// TIA Portal V20 export
DATA_BLOCK "ControlNodes"   // DB115
// stored: MemoryReserve 100, Namespace Unit1.Em7
   VAR
      em { ExternalWritable := 'False'} : "LAF_typeEmControlNode";
      cm { ExternalWritable := 'False'} : "Unit1.Em7.typeCmControlNode";
      citiMap : "LER_OEM_Data";
      conveyor { ExternalWritable := 'False'} : "Unit1.Em7.typeSequenceControlNodeConveyor";
      ngKicker { ExternalWritable := 'False'} : "Unit1.Em7.typeSequenceControlNodeNgKicker";
      passKicker { ExternalWritable := 'False'} : "Unit1.Em7.typeSequenceControlNodePassKicker";
      qrReaderSTK1 { ExternalWritable := 'False'} : "Unit1.Em7.typeSequenceControlNodeQrReadSTK1";
      qrReaderSTK2 { ExternalWritable := 'False'} : "Unit1.Em7.typeSequenceControlNodeQrReadSTK2";
      InterfaceSTK1 { ExternalWritable := 'False'} : "Unit1.Em7.typeSequenceControlNodeInterafceSTK1";
      InterfaceSTK2 { ExternalWritable := 'False'} : "Unit1.Em7.typeSequenceControlNodeInterafceSTK2";
   END_VAR
   VAR RETAIN
      cmNgKickerAxisZ { ExternalWritable := 'False'} : "LBC_typeAxisControlNode";
      cmPassKickerAxisZ { ExternalWritable := 'False'} : "LBC_typeAxisControlNode";
      cmCutConveyorAxisB { ExternalWritable := 'False'} : "LBC_typeAxisControlNode";
      cmNgConveyorAxisB { ExternalWritable := 'False'} : "LBC_typeAxisControlNode";
      cmStack1ConveyorAxisB { ExternalWritable := 'False'} : "LBC_typeAxisControlNode";
      cmStack2ConveyorAxisB { ExternalWritable := 'False'} : "LBC_typeAxisControlNode";
      cmConveyorVirtualAxisB { ExternalWritable := 'False'} : "LBC_typeAxisControlNode";
      cmCutConveyorRingBlow { ExternalWritable := 'False'} : "LBC_typeSinaSpeedControlNode";
      cmNgConveyorRingBlow { ExternalWritable := 'False'} : "LBC_typeSinaSpeedControlNode";
      cmStack2ConveyorRingBlow { ExternalWritable := 'False'} : "LBC_typeSinaSpeedControlNode";
      cmNgBoxLockCylinderUpDown { ExternalWritable := 'False'} : "LBC_typeTwoWayActuatorControlNode";
      cmNgBoxDetectSensor { ExternalWritable := 'False'} : "LBC_typeDigitalSignalControlNode";
      cmNgBoxFullSensor { ExternalWritable := 'False'} : "LBC_typeDigitalSignalControlNode";
      cmNgKickerDetectSensor { ExternalWritable := 'False'} : "LBC_typeDigitalSignalControlNode";
      cmPassKickerDetectSensor { ExternalWritable := 'False'} : "LBC_typeDigitalSignalControlNode";
      cmStack1ConveyorElectrodeDetectSensor { ExternalWritable := 'False'} : "LBC_typeDigitalSignalControlNode";
      cmStack2ConveyorElectrodeDetectSensor { ExternalWritable := 'False'} : "LBC_typeDigitalSignalControlNode";
      cmStack1QrReader { ExternalWritable := 'False'} : "LER_typeSRX300ControlNode";
      cmStack2QrReader { ExternalWritable := 'False'} : "LER_typeSRX300ControlNode";
      cmNgKickerAxisZ_TorqueCal { ExternalWritable := 'False'} : "LER_typeServoTorqueCalControlNode";
      cmPassKickerAxisZ_TorqueCal { ExternalWritable := 'False'} : "LER_typeServoTorqueCalControlNode";
      cmCutConveyorAxisB_TorqueCal { ExternalWritable := 'False'} : "LER_typeServoTorqueCalControlNode";
      cmNgConveyorAxisB_TorqueCal { ExternalWritable := 'False'} : "LER_typeServoTorqueCalControlNode";
      cmStack1ConveyorAxisB_TorqueCal { ExternalWritable := 'False'} : "LER_typeServoTorqueCalControlNode";
      cmStack2ConveyorAxisB_TorqueCal { ExternalWritable := 'False'} : "LER_typeServoTorqueCalControlNode";
   END_VAR
   VAR
      ConveyorEmpty { ExternalWritable := 'False'} : Bool;
      StackRnRCountInt { ExternalWritable := 'False'} : Int;
      StackRnRCountLReal { ExternalWritable := 'False'} : LReal;
   END_VAR
BEGIN
   // cm.brakeTest.ngKicker.monitoring.error : NG Kicker Axis Brake Test Error
   // cm.brakeTest.ngKicker.monitoring.busy : NG Kicker Axis Brake Test In progress
   // cm.brakeTest.passKicker.monitoring.error : Pass Kicker Axis Brake Test Error
   // cm.brakeTest.passKicker.monitoring.busy : Pass Kicker Axis Brake Test In progress
END_DATA_BLOCK
